// TIA Portal V20 export
DATA_BLOCK "BK17"   // DB313
// stored: MemoryReserve 100
   VAR
      "X10-1.FINAL ROLLER FRONT LIMIT SENSOR(-)" : Bool := TRUE;
      "X10-2.FINAL ROLLER FRONT HOME SENSOR" : Bool := TRUE;
      "X12-1.FINAL ROLLER FRONT LIMIT SENSOR(+)" : Bool := TRUE;
      "X12-2.SPARE" : Bool := FALSE;
      "X14-1.FINAL ROLLER REAR LIMIT SENSOR(-)" : Bool := TRUE;
      "X14-2.FINAL ROLLER REAR HOME SENSOR" : Bool := TRUE;
      "X16-1.FINAL ROLLER REAR LIMIT SENSOR(+)" : Bool := TRUE;
      "X16-2.SPARE" : Bool := FALSE;
   END_VAR
BEGIN
END_DATA_BLOCK
